PROGRAM Doff_Parallel
VAR
END_VAR

GVL.astAxes[AXIS_DOFF_PARALLEL].stInputs.bLimitBwd := TRUE;
GVL.astAxes[AXIS_DOFF_PARALLEL].stInputs.bLimitFwd := TRUE;
GVL.astAxes[AXIS_DOFF_PARALLEL].stControl.bEnable := TRUE;

END_PROGRAM

(* stored: Version 1.1.0.1, ProductVersion 3.1.4024.11
   POU Doff_Parallel: Id {9c8484c8-8761-45e8-9dcf-a9453bb68485}, SpecialFunc None *)
